(* PLC project EXAMPLE, Beckhoff Automation GmbH TwinCAT PLC Control 3.5.13.20 *)
(* stored: creationDateTime 2020-06-22T11:49:46.1535318, modificationDateTime 2020-06-22T11:49:46.1535318 *)

PROGRAM POU
VAR
	A: BOOL ;
	B: BOOL;
END_VAR

            
IF (A) THEN 
	B := FALSE;
END_IF
          
END_PROGRAM
